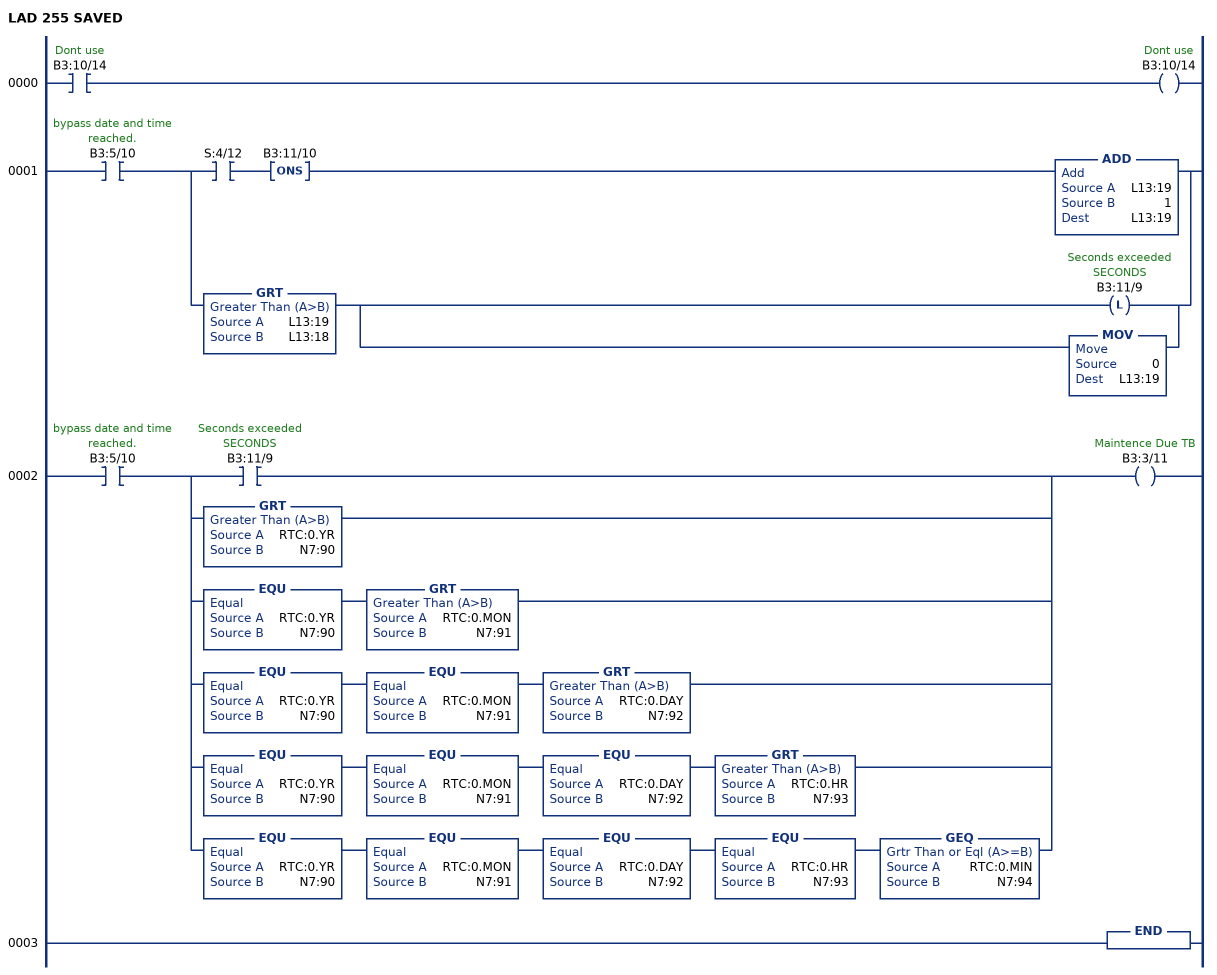
% Rung: 0 %
SOR XIC B3:10/14 OTE B3:10/14 EOR
%   B3:10/14  "Dont use" %
% Rung: 1 %
SOR XIC B3:5/10 BST XIC S:4/12 ONS B3:11/10 ADD L13:19 1 L13:19 NXB GRT L13:19 L13:18 BST OTL B3:11/9 NXB MOV 0 L13:19 BND BND EOR
%   B3:5/10  "bypass date and time reached." %
%   L13:18  MAX %
%   B3:11/9  SECONDS  "Seconds exceeded" %
% Rung: 2 %
SOR XIC B3:5/10 BST XIC B3:11/9 NXB GRT RTC:0.YR N7:90 NXB EQU RTC:0.YR N7:90 GRT RTC:0.MON N7:91 NXB EQU RTC:0.YR N7:90 EQU RTC:0.MON N7:91 GRT RTC:0.DAY N7:92 NXB EQU RTC:0.YR N7:90 EQU RTC:0.MON N7:91 EQU RTC:0.DAY N7:92 GRT RTC:0.HR N7:93 NXB EQU RTC:0.YR N7:90 EQU RTC:0.MON N7:91 EQU RTC:0.DAY N7:92 EQU RTC:0.HR N7:93 GEQ RTC:0.MIN N7:94 BND OTE B3:3/11 EOR
%   B3:5/10  "bypass date and time reached." %
%   B3:11/9  SECONDS  "Seconds exceeded" %
%   N7:90  RTC %
%   B3:3/11  TB  "Maintence Due" %
% Rung: 3 %
SOR END EOR

OTHER DOCUMENTED ADDRESSES
  B3:0/1  "toggle"
  B3:0/13  "toggle 2"
  B189:0/0  "change box"
  B189:0/9  "override boxing ok or not full signal"
  B189:0/11  "HMI force door close"
  B196:1/0  "Chute door is closed"
  B196:1/1  "control chute door"
  B196:1/13  "force box conveyor on"
  B196:3/0  "for hmi to continue production unlatched by hmi"
  HSC:0.0  "top"
  HSC:0.3/6  "Underflow interrupt"
  HSC:0.3/7  "Overflow interrupt"
  HSC:1.0  "bot"
  HSC:1.3/6  "Underflow interrupt"
  HSC:1.3/7  "Overflow interrupt"
  I:0.0/0  "Encoder Signal "A""
  I:0.0/1  "Encoder Signal "B""
  I:0.0/4  "Encoder Signal "A""
  I:0.0/5  "Encoder Signal "B""
  I:0.1/4  "not used"
  I:0.1/5  "not used"
  I:0.1/6  "not used"
  I:0.1/7  "not used"
  I:0.1/8  "not used"
  I:0.1/9  "not used"
  I:0.1/10  "not used"
  I:0.1/11  "not used"
  I:0.1/12  "not used"
  I:0.1/13  "not used"
  I:0.1/14  "not used"
  I:0.1/15  "not used"
  I:0.2  "not used"
  I:0.2/3  "Packaging Conveyor full"
  I:0.2/4  "Packaging Conveyor Box in Position"
  I:0.3  "not used"
  I:0.4  "Spare Analog Input 1"
  I:0.5  "Spare Analog Input 2"
  I:0.6  "Spare Analog Input 3"
  I:2.0/0  FRONT_ESTOP
  I:2.0/1  REAR_ESTOP
  I:2.0/8  FRONT_DOOR  "front door signal ce models only"
  I:2.0/9  REAR_DOOR  "rear door signal ce models only"
  I:2.0/11  "spare"
  L23:19  TOP_OPT_FAIL_CT
  L23:34  AIR_PRESSURE_FAULT
  L28:0  INS_1_TIME
  L29:0  INS_1_POS
  L30:0  INS_5_TIME
  L31:0  INS_5_POS
  L32:0  INS_6_TIME
  L33:0  INS_6_POS
  L192:1  BOT_LAST_TIME  "rtc bot belt previous movement event time"
  L192:2  BOT_CYCLE_TIME  "rtc bot belt time between events"
  L192:7  FROM_REAL  "distance from real part signal at optic location"
  L192:8  FROM_TRACKED  "distance from tracked part signal at optic location"
  L192:16  TOP_LAST_TIME  "rtc top belt previous movement event time"
  L192:17  TOP_CYCLE_TIME  "rtc top belt time between events"
  L199:5  ACQTM51
  L199:6  ACQTM52
  L199:7  ACQTM53
  L199:9  "ones"
  L199:10  "billions"
  L199:13  DUMP_LONG
  L199:15  ACQTM11
  L199:16  ACQTM12
  L199:17  ACQTM13
  L199:20  RESULTTM1
  L199:22  CLEARTIME5COUNT
  L199:23  CLEARTIME6COUNT
  L199:24  ACQTM61
  L199:25  ACQTM62
  L199:26  ACQTM63
  L199:27  TMSINCETRIG1
  L199:29  TMSINCETRIG5
  L199:30  TMSINCETRIG6
  L199:31  CLEARTIME1COUNT
  L199:32  RESULTTM5
  L199:33  RESULTTM6
  L199:34  MAXACQTM1
  L199:36  MAXACQTM6
  N7  
  N101:1  I2_TRIG_LOC
  N101:2  I3_TRIG_LOC
  N101:3  I4_TRIG_LOC
  O:0.0/1  "spare"
  O:0.0/11  "Spare"
  O:0.0/12  "not used"
  O:0.0/13  "not used"
  O:0.0/14  "not used"
  O:0.0/15  "not used"
  O:0.1  "not used"
  O:0.2  "not used"
  O:0.3  "not used"
  O:0.5  "spare analog output"
  O:3.0/0  "spare"
  O:3.0/2  "spare"
  O:3.0/3  "light curtain range selection /* needed? */"
  O:3.0/7  "door unlocks on CE models"
  O:3.0/8  "Light?"
  PFILE:6  "check for part jams"
  PFILE:10  "Bottom belt HSC"
  PFILE:12  "Top belt HSC"
  Q2:55  END_OF_MAIN
  Q5:94  END_OF_BELTS
  T20:0  "Trigger On Time"
  U:9  "slow data"
  U:24  "check skipped fail rate"
  U:28  "faults"
  U:29  "speed"
  U:30  "count"
  U:31  "rate calc"
  U:32  "boxer"
  U:33  "bulk pack"
  U:34  "customer boxing unit signals"
  U:35  "cleanup"

COMMENTS NOT ATTACHED TO A CURRENT RUNG
  R6:2: B41 is the top good 3 file
  R6:0: B36 is the bottom GOOD file
  R6:10: B37 is the top good 1 file
  R6:6: B35 is the top NG file
  R6:4: B34 is the bottom NG file

REVISION NOTES
  13: updated count reset
  14: added io moduals
  15: multiple steps toward new hmi integration
  21: test
  27: fix error if bulk pack and no boxing fallout were on

DATA TABLE (non-zero values as saved)
DATA B3
% B3:0 % 0X8020 0X0141 0X4001 0X9109 0X0EE5 0X0524 0X0C10 0X0421 0X3F80 0X24B0
% B3:10 % 0X2014 0X00C6 0X0000 0X8000 0X0000 0X0000 0X0000 0X0000 0X0000 0X0000
% B3:50 % 0X0001 0X0000 0X0000 0X0000 0X0000 0X0000 0X0000 0X0000 0X0000 0X0000
DATA T4
% .PRE .ACC %
% T4:0 % 0 3
% T4:1 % 150 0
% T4:2 % 400 0
% T4:3 % 222 0
% T4:4 % 1000 0
% T4:5 % 5 5
% T4:6 % 10 10
% T4:7 % 150 150
% T4:8 % 20 15
% T4:9 % 50 11
% T4:10 % 200 200
% T4:11 % 111 0
% T4:12 % 20 246
% T4:13 % 250 0
% T4:14 % 666 0
% T4:15 % 1000 1001
% T4:16 % 400 0
% T4:17 % 100 53
% T4:18 % 5 0
% T4:19 % 300 0
% T4:20 % 200 0
% T4:21 % 200 0
% T4:22 % 200 0
% T4:23 % 250 0
% T4:24 % 666 0
% T4:25 % 666 0
% T4:26 % 666 0
% T4:27 % 250 0
% T4:28 % 250 0
% T4:29 % 5000 0
% T4:30 % 333 0
% T4:31 % 333 0
% T4:32 % 222 0
% T4:33 % 222 0
DATA C5
% .PRE .ACC %
% C5:0 % 32766 0
DATA R6
% .LEN .POS %
% R6:0 % 1250 0
% R6:1 % 2000 0
% R6:2 % 1050 0
% R6:3 % 1050 0
% R6:4 % 1250 0
% R6:5 % 1250 0
% R6:6 % 1713 0
% R6:7 % 16 0
% R6:8 % 1024 0
% R6:9 % 3 0
% R6:10 % 1713 0
% R6:11 % 1050 0
% R6:12 % 10 0
% R6:13 % 10 0
% R6:14 % 10 0
% R6:15 % 10 0
% R6:16 % 1713 0
% R6:17 % 1713 0
% R6:18 % 1050 0
% R6:19 % 10 0
DATA N7
% N7:0 % 17247 3 1027 300 3 0 0 0 500 43
% N7:10 % 1000 43 0 2 20 20 1000 2000 50 1050
% N7:20 % 0 4905 10 5000 222 46 0 0 48 250
% N7:30 % 666 1412 150 0 0 1239 77 8 0 8
% N7:40 % 3 16 0 16 32767 482 1235 1350 1636 0
% N7:50 % 0 0 0 16 1 1024 0 0 32766 3
% N7:60 % 1713 1713 1050 984 1034 1024 4999 5 400 400
% N7:70 % 100 200 300 400 90 190 290 390 16425 15888
% N7:80 % 0 0 1270 1275 1300 1310 31 9 0 0
% N7:90 % 2011 4 4 12 1 31 9 222 222 12
% N7:100 % 1003 90 110 100 175 25 0 0 0 0
% N7:190 % -128 27477 27605 32767 0 0 0 0 0 0
DATA F8
% F8:0 % 6
DATA L13
% L13:0 % 12164 115601 0 35054 169022
% L13:5 % 131 4210 131 131331 111
% L13:10 % 111 96816498 30832 15 90
% L13:15 % 1485129396 -2147483648 2147483647 2147483647 82058
% L13:20 % 18673444 2042071604 777 33125 100
% L13:25 % 82 2232 91700508 111 1409426104
% L13:30 % 75702387 131 60000 1097515367 444
% L13:35 % 0 79 99 -826032397 -826032328
% L13:40 % 20436 1000000000 1000000 1097515339 1409469069
% L13:45 % 1409469079 33 0 28 3523382
% L13:50 % 75660499 67188061 1409469047 0 0
% L13:55 % 75660489 75660521 16503 -826021827 -826021822
% L13:60 % 5 104 -1783954986 600 -9
% L13:65 % 100 -900 -826028267 -826028385 12
% L13:70 % 2020509574 10 118 2043600 3523382
% L13:75 % 8919967 60 100 1409469057 6
% L13:80 % 24 74 444 7 1650276
% L13:85 % 21562260 256 258 0 75660679
% L13:90 % 75660669 5 34857 5 1409469096
% L13:95 % 10 228 0 1409469103 89410
% L13:100 % 2147483647 6 900 14 5979
% L13:105 % 89410 31 2099392 4691 2099386
% L13:110 % 6 100 50 1923692887 2020509362
% L13:115 % 2020509385 23 12 2020509373 26
% L13:120 % 19 5845 50 100 10
% L13:125 % 0 2020509574 2147483647 3276500 118378789
% L13:130 % 2 2 0 99 0
% L13:135 % 0 0 21562291 5 70
% L13:140 % 0 5 36 50 50
% L13:145 % 67188168 5 5 5 32
% L13:150 % 12 20 5115990 -5115990 96816498
% L13:155 % 0 -10 0 0 4589052
% L13:160 % 27 27 24 1220 45
% L13:165 % 2020509596 2020509606 2020509596 2020509606 6706
% L13:170 % 12817 5978 5978 600 400
% L13:175 % 4 4 42 23 38
% L13:180 % -826000057 141 51510 1000000 258000000
% L13:185 % 0 1 -826000012 142 51265
% L13:190 % 256000000 0 0 0 0
DATA L19
% L19:0 % 1409426104 1409431911 1409437126 1409442330 1409448715
% L19:5 % 1409455142 1409462880 1409468857 1409350917 1409354638
% L19:10 % 1409358086 1409390096 1409395287 1409401188 1409407615
% L19:15 % 1409413759 1409420249 0 0 0
DATA L20
% L20:0 % 1409231796 1409235337 1409238797 1409242874 1409245958
% L20:5 % 1409249139 1409320855 1409324402 1409328166 1409331571
% L20:10 % 1409334896 1409338266 1409341498 1409344795 1409347963
% L20:15 % 1409351130 1409354852 1409358296 1409390306 1409395498
% L20:20 % 1409401400 1409407827 1409413970 1409420460 1409426319
% L20:25 % 1409432126 1409437341 1409442544 1409448930 1409455357
% L20:30 % 1409463091 1409469069 1409156318 1409160924 1409165173
% L20:35 % 1409168921 1409175769 1409181377 1409185356 1409189252
% L20:40 % 1409193892 1409197921 1409201720 1409205344 1409209422
% L20:45 % 1409213668 1409217503 1409221031 1409224737 1409228477
DATA L21
% L21:0 % 2020277572 2020281033 2020284416 2020288402 2020291417
% L21:5 % 2020294528 2020364669 2020368137 2020371817 2020375146
% L21:10 % 2020378397 2020381692 2020384852 2020388076 2020391174
% L21:15 % 2020394270 2020397909 2020401277 2020432577 2020437653
% L21:20 % 2020443424 2020449710 2020455717 2020462062 2020467793
% L21:25 % 2020473473 2020478572 2020483660 2020489905 2020496191
% L21:30 % 2020503751 2020509596 2020203766 2020208268 2020212422
% L21:35 % 2020216088 2020222782 2020228265 2020232154 2020235964
% L21:40 % 2020240502 2020244441 2020248156 2020251702 2020255691
% L21:45 % 2020259844 2020263593 2020267043 2020270668 2020274326
DATA L22
% L22:0 % 1409413981 1409420470 1409426329 1409432137 1409437351
% L22:5 % 1409442554 1409448941 1409455367 1409463101 1409469079
% L22:10 % 1409156328 1409160935 1409165183 1409168931 1409175779
% L22:15 % 1409181387 1409185366 1409189262 1409193902 1409197931
% L22:20 % 1409201731 1409205354 1409209433 1409213678 1409217513
% L22:25 % 1409221041 1409224747 1409228487 1409231806 1409235348
% L22:30 % 1409238807 1409242885 1409245968 1409249149 1409320865
% L22:35 % 1409324413 1409328176 1409331581 1409334906 1409338276
% L22:40 % 1409341508 1409344805 1409347973 1409351140 1409354862
% L22:45 % 1409358307 1409390316 1409395509 1409401410 1409407837
DATA L23
% L23:0 % 2020455727 2020462072 2020467803 2020473483 2020478582
% L23:5 % 2020483670 2020489915 2020496201 2020503761 2020509606
% L23:10 % 2020203776 2020208278 2020212432 2020216098 2020222792
% L23:15 % 2020228275 2020232164 2020235974 2020240512 2020244451
% L23:20 % 2020248166 2020251712 2020255701 2020259854 2020263603
% L23:25 % 2020267053 2020270678 2020274336 2020277582 2020281043
% L23:30 % 2020284426 2020288412 2020291427 2020294538 2020364679
% L23:35 % 2020368147 2020371827 2020375156 2020378407 2020381702
% L23:40 % 2020384862 2020388086 2020391184 2020394280 2020397919
% L23:45 % 2020401287 2020432587 2020437663 2020443434 2020449720
DATA L30
% L30:0 % 1097513510 1097513738 1097513967 1097514196 1097514426
% L30:5 % 1097514655 1097514883 1097515111 1097515339 1071304727
% L30:10 % 1071304952 1071305179 1071305406 1071305631 1071305859
% L30:15 % 1071306086 1071306312 1071306539 1071306765 1071306992
% L30:20 % 1071307217 1071307442 1071307668 1071307895 1071308121
% L30:25 % 1071308347 1071308573 1071308799 1071309024 1071309250
% L30:30 % 1071309476 1071429569 1071429795 1071431153 1071431379
% L30:35 % 1071431606 1088333039 1088333266 1088334623 1088334848
% L30:40 % 1088335075 1089808842 1089809070 1089810430 1089810657
% L30:45 % 1089810882 1092780028 1092791426 1092806921 1097513283
DATA L31
% L31:0 % 3522828 3522897 3522967 3523035 3523105
% L31:5 % 3523175 3523244 3523313 3523382 2077757
% L31:10 % 2077757 2077757 2077757 2077757 2077757
% L31:15 % 2077757 2077757 2077757 2077757 2077757
% L31:20 % 2077757 2077757 2077757 2077757 2077757
% L31:25 % 2077757 2077757 2077757 2077757 2077757
% L31:30 % 2077757 2077757 2077757 2077757 2077757
% L31:35 % 2077757 2077757 2077757 2077757 2077757
% L31:40 % 2077757 2077757 2077757 2077757 2077757
% L31:45 % 2077757 2091375 2094821 2099507 3522760
DATA L32
% L32:0 % 1409351108 1409354829 1409358274 1409390283 1409395476
% L32:5 % 1409401377 1409407804 1409413948 1409420437 1409426296
% L32:10 % 1409432104 1409437319 1409442521 1409448908 1409455334
% L32:15 % 1409463068 1409469047 1409156296 1409160902 1409165150
% L32:20 % 1409168899 1409175746 1409181354 1409185333 1409189229
% L32:25 % 1409193869 1409197898 1409201698 1409205322 1409209400
% L32:30 % 1409213645 1409217480 1409221009 1409224714 1409228454
% L32:35 % 1409231774 1409235315 1409238774 1409242852 1409245936
% L32:40 % 1409249116 1409320832 1409324380 1409328144 1409331549
% L32:45 % 1409334873 1409338243 1409341475 1409344772 1409347940
DATA L33
% L33:0 % 2020394248 2020397887 2020401255 2020432555 2020437631
% L33:5 % 2020443402 2020449688 2020455695 2020462040 2020467771
% L33:10 % 2020473451 2020478550 2020483638 2020489883 2020496169
% L33:15 % 2020503729 2020509574 2020203744 2020208246 2020212400
% L33:20 % 2020216066 2020222760 2020228243 2020232132 2020235942
% L33:25 % 2020240480 2020244419 2020248134 2020251680 2020255669
% L33:30 % 2020259822 2020263571 2020267021 2020270646 2020274304
% L33:35 % 2020277550 2020281011 2020284394 2020288380 2020291395
% L33:40 % 2020294506 2020364647 2020368115 2020371795 2020375124
% L33:45 % 2020378375 2020381670 2020384830 2020388054 2020391152
DATA B100
% B100:0 % 0X2780 0X18A8 0X0004 0X0000 0X0000 0X0000 0X0000 0X0000 0X0000 0X0000
DATA N101
% N101:0 % 114 0 0 0 1183 100 1015 1200 1216 1238
% N101:10 % 1248 1604 10 16383 1269 17365 3018 222 333 333
% N101:20 % 1000 500 400 0 0 0 222 222 0 0
DATA L102
% L102:0 % 20 10 4988 5000 5000
% L102:5 % 5000 0 111 0 0
% L102:10 % -5115990 114 0 0 34857
% L102:15 % 0 30 10 30 10
% L102:20 % 0 6 67755 0 27
% L102:25 % 28 0 66252844 81649 9418788
% L102:30 % 10 0 9 7746 0
% L102:35 % 174 302 0 999999 24
% L102:40 % 0 4 63154 0 0
